FUNCTION_BLOCK FB_INFLUX_DB_ADS IMPLEMENTS I_INFLUXDB_ADS
VAR_IN_OUT
  bResult:                                                BOOL;
END_VAR
VAR_INPUT
  bADSLifeBit:                                            BOOL;
  bAdsConnected:                                          BOOL;
  bReady:                                                 BOOL;
  bBusy:                                                  BOOL;
END_VAR
VAR //General
	{attribute 'instance-path'} 
  {attribute 'noinit'} 
	strInstancePath:									                      STRING;
	bInit: 												                          BOOL:=TRUE;
	strFullObjectPath: 								                      STRING;
	stEvent:											                          ST_EVENT;
	bAck:												                            BOOL;
	
END_VAR
VAR   // From FB_init	
	itfOpMode:											                        I_OP_MODE; 
  itfEventLogger:                                         I_EVENT_LOGGER;
END_VAR                                      				
VAR	// Step chain control                				
  eSeq, eLastSeq, eNextSeq:					                      E_SEQ_DATABASE; 
  i:														                          INT;
  stSeqCtrlGeneral:											                  ST_SEQ_CTRL_GEN;     	
END_VAR                                             		
VAR                                                 		
	bMethodeFromExtStarted:									                BOOL;
	bMethodeFromExtActive:									                BOOL;
	bMethodeFromExtDone:									                  BOOL;
	strTemp:												                        STRING;
END_VAR   
VAR
  // From ADS
  bDBLifeBit:                                             BOOL;
  liDatabaseSizeInMb:                                     LINT;
  udiDatabaseSizeInMb:                                    UDINT;
  uiTotalMeasurements:                                    UINT;
  // To ADS
  bGetBucketExist:                                        BOOL;
  sBucketName:                                            T_MaxString := '3925-HZP';
  bGetMeasurementExist:                                   BOOL;
  sMeasurementName:                                       T_MaxString;
  bDeleteMeasurement:                                     BOOL;
  bDeleteAllMeasurements:                                 BOOL;
  bWriteStructData:                                       BOOL;
  sTagName:                                               T_MaxString;
  sFieldName:                                             T_MaxString;
  stFieldValues:                                          ST_DATABASE_RECORD;
  pFieldStructContent:                                    POINTER TO ARRAY [0..99] OF T_MaxString;
  pFieldNames:                                            POINTER TO ARRAY [0..99] OF T_MaxString;
  dtFrom:                                                 DT;
  dtTo:                                                   DT;
  sDtFrom:                                                T_MaxString;
  sDtTo:                                                  T_MaxString;
  sFieldNameExistCheck:                                   T_MaxString;
  bGetTagExist:                                           BOOL;
  bGetFieldExist:                                         BOOL;
  bClearMeasurement:                                      BOOL;
  bDeleteTag:                                             BOOL;
  bDeleteTagContentBlock:                                 BOOL;
  bDeleteField:                                           BOOL;
  bGetTotalMeasurements:                                  BOOL;
END_VAR    
VAR // State
  tLifeBitTimeout:                                        TIME := T#5S;
  // ADS
  uiADSStateSeq:                                          UINT := 0;
  tonADSState:                                            TON;
  bResetADSStateTimer:                                    BOOL;
  bADSState:                                              BOOL := TRUE;
  // InfluxDB
  uiInfluxDBStateSeq:                                     UINT := 0;
  tonInfluxDBState:                                       TON;
  bResetInfluxDBStateTimer:                               BOOL;
  bInfluxDBState:                                         BOOL := TRUE;
END_VAR              	
VAR_TEMP                    	
	iTemp:										                              INT;
END_VAR

// Set FBs and Interfaces ready after switch internal step
IF stSeqCtrlGeneral.iInternalSeqStateCase <> stSeqCtrlGeneral.iLastInternalSeqStateCase AND NOT stSeqCtrlGeneral.bExitSetReadyState THEN
  IF TRUE
  THEN
    stSeqCtrlGeneral.bExitSetReadyState := TRUE;
  ELSE
    RETURN;
  END_IF
END_IF

stSeqCtrlGeneral.strObject := F_CreateObjectName(strInstancePath);

// Init
// Format Time string for InfluxDB
sDtFrom := DT_TO_STRING(dtFrom);
sDtFrom := DELETE(sDtFrom, 3, 1);
sDtFrom := REPLACE(sDtFrom, 'T', 1, 11);
sDtFrom := CONCAT(sDtFrom, 'Z');
sDtTo := DT_TO_STRING(dtTo);
sDtTo := DELETE(sDtTo, 3, 1);
sDtTo := REPLACE(sDtTo, 'T', 1, 11);
sDtTo := CONCAT(sDtTo, 'Z');

// Actions
A_010_ADSState();
A_020_InfluxDBState();

// First method call
_m_SequenceManager();
//_m_SaveLastStep();

udiDatabaseSizeInMb := TO_UDINT(liDatabaseSizeInMb);

CASE eSeq OF 
  E_SEQ_DATABASE.BASE:;
  
	E_SEQ_DATABASE.INIT: _m_Seq_INIT();
		IF TRUE
		AND (stSeqCtrlGeneral.eActiveSeqState = E_SEQ_GENERAL.DONE) 
		THEN
			eSeq := E_SEQ_DATABASE.BASE;
		END_IF
		
	E_SEQ_DATABASE.SETUP:;
  
	// Process
  E_SEQ_DATABASE.BUCKET_EXIST_CHECK: _m_Seq_BUCKET_EXIST_CHECK();
    IF TRUE
		AND (stSeqCtrlGeneral.eActiveSeqState = E_SEQ_GENERAL.DONE) 
		THEN
			eSeq := E_SEQ_DATABASE.BASE;
		END_IF
  
	E_SEQ_DATABASE.MEASUREMENT_EXIST_CHECK:         _m_Seq_MEASUREMENT_EXIST_CHECK();
    IF TRUE
		AND (stSeqCtrlGeneral.eActiveSeqState = E_SEQ_GENERAL.DONE) 
		THEN
			eSeq := E_SEQ_DATABASE.BASE;
		END_IF
    
  E_SEQ_DATABASE.WRITE_STRUCT:  _m_Seq_WRITE_STRUCT();
    IF TRUE
		AND (stSeqCtrlGeneral.eActiveSeqState = E_SEQ_GENERAL.DONE) 
		THEN
			eSeq := E_SEQ_DATABASE.BASE;
		END_IF
  
  E_SEQ_DATABASE.TAG_EXIST_CHECK:     _m_Seq_TAG_EXIST_CHECK();
    IF TRUE
		AND (stSeqCtrlGeneral.eActiveSeqState = E_SEQ_GENERAL.DONE) 
		THEN
			eSeq := E_SEQ_DATABASE.BASE;
		END_IF
    
  E_SEQ_DATABASE.FIELD_EXIST_CHECK:     _m_Seq_FIELD_EXIST_CHECK();
    IF TRUE
		AND (stSeqCtrlGeneral.eActiveSeqState = E_SEQ_GENERAL.DONE) 
		THEN
			eSeq := E_SEQ_DATABASE.BASE;
		END_IF
    
  E_SEQ_DATABASE.DELETE_MEASUREMENT:    _m_Seq_DELETE_MEASUREMENT();
    IF TRUE
		AND (stSeqCtrlGeneral.eActiveSeqState = E_SEQ_GENERAL.DONE) 
		THEN
			eSeq := E_SEQ_DATABASE.BASE;
		END_IF
    
  E_SEQ_DATABASE.DELETE_ALL_MEASUREMENTS:    _m_Seq_DELETE_ALL_MEASUREMENTS();
    IF TRUE
		AND (stSeqCtrlGeneral.eActiveSeqState = E_SEQ_GENERAL.DONE) 
		THEN
			eSeq := E_SEQ_DATABASE.BASE;
		END_IF
  
  E_SEQ_DATABASE.DELETE_TAG:    _m_Seq_DELETE_TAG();
    IF TRUE
		AND (stSeqCtrlGeneral.eActiveSeqState = E_SEQ_GENERAL.DONE) 
		THEN
			eSeq := E_SEQ_DATABASE.BASE;
		END_IF
    
  E_SEQ_DATABASE.DELETE_TAG_CONTENT_BLOCK:    _m_Seq_DELETE_TAG_CONTENT_BLOCK();
    IF TRUE
		AND (stSeqCtrlGeneral.eActiveSeqState = E_SEQ_GENERAL.DONE) 
		THEN
			eSeq := E_SEQ_DATABASE.BASE;
		END_IF
  
  E_SEQ_DATABASE.DELETE_FIELD:           _m_Seq_DELETE_FIELD();
    IF TRUE
		AND (stSeqCtrlGeneral.eActiveSeqState = E_SEQ_GENERAL.DONE) 
		THEN
			eSeq := E_SEQ_DATABASE.BASE;
		END_IF
    
  E_SEQ_DATABASE.GET_TOTAL_MEASUREMENTS:           _m_Seq_GET_TOTAL_MEASUREMENTS();
    IF TRUE
		AND (stSeqCtrlGeneral.eActiveSeqState = E_SEQ_GENERAL.DONE) 
		THEN
			eSeq := E_SEQ_DATABASE.BASE;
		END_IF

  // End
	E_SEQ_DATABASE.END:;
	E_SEQ_DATABASE.ERROR_SEQ:;	
END_CASE

strTemp:=TO_STRING(eSeq);

METHOD PRIVATE _m_DebugManager
VAR_INPUT
	iStepID: int;
END_VAR
IF TRUE
AND THIS^.stSeqCtrlGeneral.bDebugModeActive 
AND NOT THIS^.stSeqCtrlGeneral.bActiveStep
THEN


THIS^.stSeqCtrlGeneral.bBreakpointActive:=FALSE;

FOR i:=0 TO 10 DO
	
	IF TRUE
	AND iStepID=THIS^.stSeqCtrlGeneral.listBreakpoint[i] 
	AND iStepID<>0
	THEN
		EXIT;
	END_IF
END_FOR
IF (i<=10) THEN
	THIS^.stSeqCtrlGeneral.bBreakpointActive:=TRUE;
END_IF

END_IF
END_METHOD

METHOD PRIVATE _m_Delay : BOOL
VAR_INPUT
	DelayTime:	TIME;
END_VAR
THIS^.stSeqCtrlGeneral.bDelayActive:=TRUE;
THIS^.stSeqCtrlGeneral.tDelay:=DelayTime;
_m_Delay:=FALSE;
IF THIS^.stSeqCtrlGeneral.tonDelay.Q THEN
	_m_Delay:=TRUE;
END_IF
END_METHOD

METHOD PRIVATE _m_GeneralStepSetting : BOOL
VAR_INPUT
	StepType:			    	E_STEP_STATE_TYPE;
	InfoTextID:					STRING(20);
	EnableDebug:	   			BOOL;	
	
END_VAR
IF THIS^.stSeqCtrlGeneral.bActiveStep THEN
	THIS^.stSeqCtrlGeneral.eStep_Type:=StepType;
	THIS^.stSeqCtrlGeneral.strExtraInfo:= GenLib.F_RET_TXTLIST_ENTRY(strPortNr:='851',strID:='',strTxtLstName:=InfoTextID);
END_IF
END_METHOD

METHOD PRIVATE _m_SaveLastStep : BOOL
VAR_INPUT
END_VAR
VAR
	i: dint;
END_VAR
IF NOT THIS^.stSeqCtrlGeneral.bActiveStep THEN
	
	FOR i:=49 TO 1 BY -1 DO
			stSeqCtrlGeneral.listLastSteps[i].strStepName:=stSeqCtrlGeneral.listLastSteps[i-1].strStepName;
			stSeqCtrlGeneral.listLastSteps[i].tStepTime:=stSeqCtrlGeneral.listLastSteps[i-1].tStepTime;
			stSeqCtrlGeneral.listLastSteps[i].tDelayTime:=stSeqCtrlGeneral.listLastSteps[i-1].tDelayTime;
	END_FOR
	stSeqCtrlGeneral.listLastSteps[0].strStepName:=TO_STRING(THIS^.eSeq);
	stSeqCtrlGeneral.listLastSteps[1].tStepTime:=THIS^.stSeqCtrlGeneral.tonStepTime.ET;
	stSeqCtrlGeneral.listLastSteps[1].tStepTime:=THIS^.stSeqCtrlGeneral.tonDelay.ET;
ELSE
	stSeqCtrlGeneral.listLastSteps[0].tStepTime:=THIS^.stSeqCtrlGeneral.tonStepTime.ET;
	stSeqCtrlGeneral.listLastSteps[0].tDelayTime:=THIS^.stSeqCtrlGeneral.tonDelay.ET;	
END_IF
END_METHOD

METHOD PRIVATE _m_Seq_BUCKET_EXIST_CHECK : E_SEQ_PROCESS
VAR_INPUT
END_VAR
VAR
	ActiveSeq: STRING;
END_VAR
//THIS^._m_GeneralStepSetting(StepType:=E_STEP_STATE_TYPE.INIT,
ActiveSeq := TO_STRING(THIS^.eSeq);

CASE THIS^.stSeqCtrlGeneral.eActiveSeqState OF
E_SEQ_GENERAL.READY:;
	
E_SEQ_GENERAL.EXECUTE:;
	IF TRUE
	THEN
		THIS^.stSeqCtrlGeneral.eActiveSeqState := E_SEQ_GENERAL.RESET;
	END_IF
  
E_SEQ_GENERAL.RESET:;
	THIS^.stSeqCtrlGeneral.iInternalSeqStateCase := 0;
	IF TRUE
	THEN
    THIS^.bResult := FALSE;
		THIS^.stSeqCtrlGeneral.eActiveSeqState := E_SEQ_GENERAL.BUSY;
	END_IF
  
E_SEQ_GENERAL.BUSY:;
	CASE THIS^.stSeqCtrlGeneral.iInternalSeqStateCase OF
    0:  // Execute
      IF TRUE 
      AND THIS^.bAdsConnected
      AND NOT THIS^.bBusy
      AND THIS^.bReady
			THEN 
        THIS^.bGetBucketExist := TRUE;
        THIS^.stSeqCtrlGeneral.iInternalSeqStateCase := 10;
			END_IF

    10:	// Wait for done
      IF TRUE 
      AND NOT THIS^.bBusy
      AND THIS^.bReady
      AND NOT THIS^.bGetBucketExist
			THEN 
        THIS^.stSeqCtrlGeneral.iInternalSeqStateCase := 1000;
			END_IF
      
    1000: // Exit step
      IF TRUE
      THEN
        THIS^.stSeqCtrlGeneral.iInternalSeqStateCase := 9999;
			END_IF
      
	ELSE
		THIS^.stSeqCtrlGeneral.eActiveSeqState := E_SEQ_GENERAL.DONE;  
	END_CASE
	THIS^.stSeqCtrlGeneral.strExtraInfo := CONCAT('Internal state: ', TO_STRING(THIS^.stSeqCtrlGeneral.iInternalSeqStateCase));

E_SEQ_GENERAL.DONE:;

E_SEQ_GENERAL.ERROR:;

E_SEQ_GENERAL.TIME_OUT:; 

ELSE
  THIS^.stSeqCtrlGeneral.eActiveSeqState := E_SEQ_GENERAL.ERROR;
END_CASE
END_METHOD

METHOD PRIVATE _m_Seq_CLEAR_MEASUREMENT : E_SEQ_PROCESS
VAR_INPUT
END_VAR
VAR
	ActiveSeq: STRING;
END_VAR
//THIS^._m_GeneralStepSetting(StepType:=E_STEP_STATE_TYPE.INIT,
ActiveSeq := TO_STRING(THIS^.eSeq);

CASE THIS^.stSeqCtrlGeneral.eActiveSeqState OF
E_SEQ_GENERAL.READY:;
	
E_SEQ_GENERAL.EXECUTE:;
	IF TRUE
	THEN
		THIS^.stSeqCtrlGeneral.eActiveSeqState := E_SEQ_GENERAL.RESET;
	END_IF
  
E_SEQ_GENERAL.RESET:;
	THIS^.stSeqCtrlGeneral.iInternalSeqStateCase := 0;
	IF TRUE
	THEN
    THIS^.bResult := FALSE;
		THIS^.stSeqCtrlGeneral.eActiveSeqState := E_SEQ_GENERAL.BUSY;
	END_IF
  
E_SEQ_GENERAL.BUSY:;
	CASE THIS^.stSeqCtrlGeneral.iInternalSeqStateCase OF
		0:	// Entrance step --> Create command
      IF TRUE 
      AND THIS^.bAdsConnected
      AND NOT THIS^.bBusy
      AND THIS^.bReady
			THEN 
        THIS^.bClearMeasurement := TRUE;
        THIS^.stSeqCtrlGeneral.iInternalSeqStateCase := 10;
			END_IF
      
    10:	// Wait for done
      IF TRUE 
      AND NOT THIS^.bBusy
      AND THIS^.bReady
      AND NOT THIS^.bClearMeasurement
			THEN 
        THIS^.stSeqCtrlGeneral.iInternalSeqStateCase := 1000;
			END_IF
      
    1000: // Exit step
      IF TRUE
      THEN
        THIS^.stSeqCtrlGeneral.iInternalSeqStateCase := 9999;
			END_IF
      
	ELSE
		THIS^.stSeqCtrlGeneral.eActiveSeqState := E_SEQ_GENERAL.DONE;  
	END_CASE
	THIS^.stSeqCtrlGeneral.strExtraInfo := CONCAT('Internal state: ', TO_STRING(THIS^.stSeqCtrlGeneral.iInternalSeqStateCase));

E_SEQ_GENERAL.DONE:;

E_SEQ_GENERAL.ERROR:;

E_SEQ_GENERAL.TIME_OUT:; 
IF TRUE
AND THIS^.stSeqCtrlGeneral.bTimeOutActiveQuit 
THEN
  THIS^.stSeqCtrlGeneral.strExtraInfo := 'Bitte quittieren und erneut testen';
  IF TRUE
  //AND itfOpMode.P_QUIT
  THEN
    THIS^.stSeqCtrlGeneral.eActiveSeqState := E_SEQ_GENERAL.EXECUTE;
	END_IF
  
END_IF

ELSE
  THIS^.stSeqCtrlGeneral.eActiveSeqState := E_SEQ_GENERAL.ERROR;
END_CASE
END_METHOD

METHOD PRIVATE _m_Seq_DELETE_ALL_MEASUREMENTS : E_SEQ_PROCESS
VAR_INPUT
END_VAR
VAR
	ActiveSeq: STRING;
END_VAR
//THIS^._m_GeneralStepSetting(StepType:=E_STEP_STATE_TYPE.INIT,
ActiveSeq := TO_STRING(THIS^.eSeq);

CASE THIS^.stSeqCtrlGeneral.eActiveSeqState OF
E_SEQ_GENERAL.READY:;

E_SEQ_GENERAL.EXECUTE:;
	IF TRUE
	THEN
		THIS^.stSeqCtrlGeneral.eActiveSeqState := E_SEQ_GENERAL.RESET;
	END_IF
  
E_SEQ_GENERAL.RESET:;
	THIS^.stSeqCtrlGeneral.iInternalSeqStateCase := 0;
	IF TRUE
	THEN
    THIS^.bResult := FALSE;
		THIS^.stSeqCtrlGeneral.eActiveSeqState := E_SEQ_GENERAL.BUSY;
	END_IF
  
E_SEQ_GENERAL.BUSY:;
	CASE THIS^.stSeqCtrlGeneral.iInternalSeqStateCase OF
		0:	// Entrance step --> Create command
      IF TRUE 
      AND THIS^.bAdsConnected
      AND NOT THIS^.bBusy
      AND THIS^.bReady
			THEN 
        THIS^.bDeleteAllMeasurements := TRUE;
        THIS^.stSeqCtrlGeneral.iInternalSeqStateCase := 10;
			END_IF
      
    10:	// Wait for done
      IF TRUE 
      AND NOT THIS^.bBusy
      AND THIS^.bReady
      AND NOT THIS^.bDeleteAllMeasurements
			THEN 
        THIS^.stSeqCtrlGeneral.iInternalSeqStateCase := 1000;
			END_IF
      
    1000: // Exit step
      IF TRUE
      THEN
        THIS^.stSeqCtrlGeneral.iInternalSeqStateCase := 9999;
			END_IF
      
	ELSE
		THIS^.stSeqCtrlGeneral.eActiveSeqState := E_SEQ_GENERAL.DONE;  
	END_CASE
	THIS^.stSeqCtrlGeneral.strExtraInfo := CONCAT('Internal state: ', TO_STRING(THIS^.stSeqCtrlGeneral.iInternalSeqStateCase));

E_SEQ_GENERAL.DONE:;

E_SEQ_GENERAL.ERROR:;

E_SEQ_GENERAL.TIME_OUT:; 
IF TRUE
AND THIS^.stSeqCtrlGeneral.bTimeOutActiveQuit 
THEN
  THIS^.stSeqCtrlGeneral.strExtraInfo := 'Bitte quittieren und erneut testen';
  IF TRUE
  //AND itfOpMode.P_QUIT
  THEN
    THIS^.stSeqCtrlGeneral.eActiveSeqState := E_SEQ_GENERAL.EXECUTE;
	END_IF
  
END_IF

ELSE
  THIS^.stSeqCtrlGeneral.eActiveSeqState := E_SEQ_GENERAL.ERROR;
END_CASE
END_METHOD

METHOD PRIVATE _m_Seq_DELETE_FIELD : E_SEQ_PROCESS
VAR_INPUT
END_VAR
VAR
	ActiveSeq: STRING;
END_VAR
//THIS^._m_GeneralStepSetting(StepType:=E_STEP_STATE_TYPE.INIT,
ActiveSeq := TO_STRING(THIS^.eSeq);

CASE THIS^.stSeqCtrlGeneral.eActiveSeqState OF
E_SEQ_GENERAL.READY:;
	
E_SEQ_GENERAL.EXECUTE:;
	IF TRUE
	THEN
		THIS^.stSeqCtrlGeneral.eActiveSeqState := E_SEQ_GENERAL.RESET;
	END_IF
  
E_SEQ_GENERAL.RESET:;
	THIS^.stSeqCtrlGeneral.iInternalSeqStateCase := 0;
	IF TRUE
	THEN
    THIS^.bResult := FALSE;
		THIS^.stSeqCtrlGeneral.eActiveSeqState := E_SEQ_GENERAL.BUSY;
	END_IF
  
E_SEQ_GENERAL.BUSY:;
	CASE THIS^.stSeqCtrlGeneral.iInternalSeqStateCase OF
    0:  // Execute
      IF TRUE 
      AND THIS^.bAdsConnected
      AND NOT THIS^.bBusy
      AND THIS^.bReady
			THEN 
        THIS^.bDeleteField := TRUE;
        THIS^.stSeqCtrlGeneral.iInternalSeqStateCase := 10;
			END_IF

    10:	// Wait for done
      IF TRUE 
      AND NOT THIS^.bBusy
      AND THIS^.bReady
      AND NOT THIS^.bDeleteField
			THEN 
        THIS^.stSeqCtrlGeneral.iInternalSeqStateCase := 1000;
			END_IF
      
    1000: // Exit step
      IF TRUE
      THEN
        THIS^.stSeqCtrlGeneral.iInternalSeqStateCase := 9999;
			END_IF
      
	ELSE
		THIS^.stSeqCtrlGeneral.eActiveSeqState := E_SEQ_GENERAL.DONE;  
	END_CASE
	THIS^.stSeqCtrlGeneral.strExtraInfo := CONCAT('Internal state: ', TO_STRING(THIS^.stSeqCtrlGeneral.iInternalSeqStateCase));

E_SEQ_GENERAL.DONE:;

E_SEQ_GENERAL.ERROR:;

E_SEQ_GENERAL.TIME_OUT:; 

ELSE
  THIS^.stSeqCtrlGeneral.eActiveSeqState := E_SEQ_GENERAL.ERROR;
END_CASE
END_METHOD

METHOD PRIVATE _m_Seq_DELETE_MEASUREMENT : E_SEQ_PROCESS
VAR_INPUT
END_VAR
VAR
	ActiveSeq: STRING;
END_VAR
//THIS^._m_GeneralStepSetting(StepType:=E_STEP_STATE_TYPE.INIT,
ActiveSeq := TO_STRING(THIS^.eSeq);

CASE THIS^.stSeqCtrlGeneral.eActiveSeqState OF
E_SEQ_GENERAL.READY:;
	
E_SEQ_GENERAL.EXECUTE:;
	IF TRUE
	THEN
		THIS^.stSeqCtrlGeneral.eActiveSeqState := E_SEQ_GENERAL.RESET;
	END_IF
  
E_SEQ_GENERAL.RESET:;
	THIS^.stSeqCtrlGeneral.iInternalSeqStateCase := 0;
	IF TRUE
	THEN
    THIS^.bResult := FALSE;
		THIS^.stSeqCtrlGeneral.eActiveSeqState := E_SEQ_GENERAL.BUSY;
	END_IF
  
E_SEQ_GENERAL.BUSY:;
	CASE THIS^.stSeqCtrlGeneral.iInternalSeqStateCase OF
		0:	// Entrance step --> Create command
      IF TRUE 
      AND THIS^.bAdsConnected
      AND NOT THIS^.bBusy
      AND THIS^.bReady
			THEN 
        THIS^.bDeleteMeasurement := TRUE;
        THIS^.stSeqCtrlGeneral.iInternalSeqStateCase := 10;
			END_IF
      
    10:	// Wait for done
      IF TRUE 
      AND NOT THIS^.bBusy
      AND THIS^.bReady
      AND NOT THIS^.bDeleteMeasurement
			THEN 
        THIS^.stSeqCtrlGeneral.iInternalSeqStateCase := 1000;
			END_IF
      
    1000: // Exit step
      IF TRUE
      THEN
        THIS^.stSeqCtrlGeneral.iInternalSeqStateCase := 9999;
			END_IF
      
	ELSE
		THIS^.stSeqCtrlGeneral.eActiveSeqState := E_SEQ_GENERAL.DONE;  
	END_CASE
	THIS^.stSeqCtrlGeneral.strExtraInfo := CONCAT('Internal state: ', TO_STRING(THIS^.stSeqCtrlGeneral.iInternalSeqStateCase));

E_SEQ_GENERAL.DONE:;

E_SEQ_GENERAL.ERROR:;

E_SEQ_GENERAL.TIME_OUT:; 
IF TRUE
AND THIS^.stSeqCtrlGeneral.bTimeOutActiveQuit 
THEN
  THIS^.stSeqCtrlGeneral.strExtraInfo := 'Bitte quittieren und erneut testen';
  IF TRUE
  //AND itfOpMode.P_QUIT
  THEN
    THIS^.stSeqCtrlGeneral.eActiveSeqState := E_SEQ_GENERAL.EXECUTE;
	END_IF
  
END_IF

ELSE
  THIS^.stSeqCtrlGeneral.eActiveSeqState := E_SEQ_GENERAL.ERROR;
END_CASE
END_METHOD

METHOD PRIVATE _m_Seq_DELETE_TAG : E_SEQ_PROCESS
VAR_INPUT
END_VAR
VAR
	ActiveSeq: STRING;
END_VAR
//THIS^._m_GeneralStepSetting(StepType:=E_STEP_STATE_TYPE.INIT,
ActiveSeq := TO_STRING(THIS^.eSeq);

CASE THIS^.stSeqCtrlGeneral.eActiveSeqState OF
E_SEQ_GENERAL.READY:;
	
E_SEQ_GENERAL.EXECUTE:;
	IF TRUE
	THEN
		THIS^.stSeqCtrlGeneral.eActiveSeqState := E_SEQ_GENERAL.RESET;
	END_IF
  
E_SEQ_GENERAL.RESET:;
	THIS^.stSeqCtrlGeneral.iInternalSeqStateCase := 0;
	IF TRUE
	THEN
    THIS^.bResult := FALSE;
		THIS^.stSeqCtrlGeneral.eActiveSeqState := E_SEQ_GENERAL.BUSY;
	END_IF
  
E_SEQ_GENERAL.BUSY:;
	CASE THIS^.stSeqCtrlGeneral.iInternalSeqStateCase OF
    0:  // Execute
      IF TRUE 
      AND THIS^.bAdsConnected
      AND NOT THIS^.bBusy
      AND THIS^.bReady
			THEN 
        THIS^.bDeleteTag := TRUE;
        THIS^.stSeqCtrlGeneral.iInternalSeqStateCase := 10;
			END_IF

    10:	// Wait for done
      IF TRUE 
      AND NOT THIS^.bBusy
      AND THIS^.bReady
      AND NOT THIS^.bDeleteTag
			THEN 
        THIS^.stSeqCtrlGeneral.iInternalSeqStateCase := 1000;
			END_IF
      
    1000: // Exit step
      IF TRUE
      THEN
        THIS^.stSeqCtrlGeneral.iInternalSeqStateCase := 9999;
			END_IF
      
	ELSE
		THIS^.stSeqCtrlGeneral.eActiveSeqState := E_SEQ_GENERAL.DONE;  
	END_CASE
	THIS^.stSeqCtrlGeneral.strExtraInfo := CONCAT('Internal state: ', TO_STRING(THIS^.stSeqCtrlGeneral.iInternalSeqStateCase));

E_SEQ_GENERAL.DONE:;

E_SEQ_GENERAL.ERROR:;

E_SEQ_GENERAL.TIME_OUT:; 

ELSE
  THIS^.stSeqCtrlGeneral.eActiveSeqState := E_SEQ_GENERAL.ERROR;
END_CASE
END_METHOD

METHOD PRIVATE _m_Seq_DELETE_TAG_CONTENT_BLOCK : E_SEQ_PROCESS
VAR_INPUT
END_VAR
VAR
	ActiveSeq: STRING;
END_VAR
//THIS^._m_GeneralStepSetting(StepType:=E_STEP_STATE_TYPE.INIT,
ActiveSeq := TO_STRING(THIS^.eSeq);

CASE THIS^.stSeqCtrlGeneral.eActiveSeqState OF
E_SEQ_GENERAL.READY:;
	
E_SEQ_GENERAL.EXECUTE:;
	IF TRUE
	THEN
		THIS^.stSeqCtrlGeneral.eActiveSeqState := E_SEQ_GENERAL.RESET;
	END_IF
  
E_SEQ_GENERAL.RESET:;
	THIS^.stSeqCtrlGeneral.iInternalSeqStateCase := 0;
	IF TRUE
	THEN
    THIS^.bResult := FALSE;
		THIS^.stSeqCtrlGeneral.eActiveSeqState := E_SEQ_GENERAL.BUSY;
	END_IF
  
E_SEQ_GENERAL.BUSY:;
	CASE THIS^.stSeqCtrlGeneral.iInternalSeqStateCase OF
    0:  // Execute
      IF TRUE 
      AND THIS^.bAdsConnected
      AND NOT THIS^.bBusy
      AND THIS^.bReady
			THEN 
        THIS^.bDeleteTagContentBlock := TRUE;
        THIS^.stSeqCtrlGeneral.iInternalSeqStateCase := 10;
			END_IF

    10:	// Wait for done
      IF TRUE 
      AND NOT THIS^.bBusy
      AND THIS^.bReady
      AND NOT THIS^.bDeleteTagContentBlock
			THEN 
        THIS^.stSeqCtrlGeneral.iInternalSeqStateCase := 1000;
			END_IF
      
    1000: // Exit step
      IF TRUE
      THEN
        THIS^.stSeqCtrlGeneral.iInternalSeqStateCase := 9999;
			END_IF
      
	ELSE
		THIS^.stSeqCtrlGeneral.eActiveSeqState := E_SEQ_GENERAL.DONE;  
	END_CASE
	THIS^.stSeqCtrlGeneral.strExtraInfo := CONCAT('Internal state: ', TO_STRING(THIS^.stSeqCtrlGeneral.iInternalSeqStateCase));

E_SEQ_GENERAL.DONE:;

E_SEQ_GENERAL.ERROR:;

E_SEQ_GENERAL.TIME_OUT:; 

ELSE
  THIS^.stSeqCtrlGeneral.eActiveSeqState := E_SEQ_GENERAL.ERROR;
END_CASE
END_METHOD

METHOD PRIVATE _m_Seq_FIELD_EXIST_CHECK : E_SEQ_PROCESS
VAR_INPUT
END_VAR
VAR
	ActiveSeq: STRING;
END_VAR
//THIS^._m_GeneralStepSetting(StepType:=E_STEP_STATE_TYPE.INIT,
ActiveSeq := TO_STRING(THIS^.eSeq);

CASE THIS^.stSeqCtrlGeneral.eActiveSeqState OF
E_SEQ_GENERAL.READY:;
	
E_SEQ_GENERAL.EXECUTE:;
	IF TRUE
	THEN
		THIS^.stSeqCtrlGeneral.eActiveSeqState := E_SEQ_GENERAL.RESET;
	END_IF
  
E_SEQ_GENERAL.RESET:;
	THIS^.stSeqCtrlGeneral.iInternalSeqStateCase := 0;
	IF TRUE
	THEN
    THIS^.bResult := FALSE;
		THIS^.stSeqCtrlGeneral.eActiveSeqState := E_SEQ_GENERAL.BUSY;
	END_IF
  
E_SEQ_GENERAL.BUSY:;
	CASE THIS^.stSeqCtrlGeneral.iInternalSeqStateCase OF
    0:  // Execute
      IF TRUE 
      AND THIS^.bAdsConnected
      AND NOT THIS^.bBusy
      AND THIS^.bReady
			THEN 
        THIS^.bGetFieldExist := TRUE;
        THIS^.stSeqCtrlGeneral.iInternalSeqStateCase := 10;
			END_IF

    10:	// Wait for done
      IF TRUE 
      AND NOT THIS^.bBusy
      AND THIS^.bReady
      AND NOT THIS^.bGetFieldExist
			THEN 
        THIS^.stSeqCtrlGeneral.iInternalSeqStateCase := 1000;
			END_IF
      
    1000: // Exit step
      IF TRUE
      THEN
        THIS^.stSeqCtrlGeneral.iInternalSeqStateCase := 9999;
			END_IF
      
	ELSE
		THIS^.stSeqCtrlGeneral.eActiveSeqState := E_SEQ_GENERAL.DONE;  
	END_CASE
	THIS^.stSeqCtrlGeneral.strExtraInfo := CONCAT('Internal state: ', TO_STRING(THIS^.stSeqCtrlGeneral.iInternalSeqStateCase));

E_SEQ_GENERAL.DONE:;

E_SEQ_GENERAL.ERROR:;

E_SEQ_GENERAL.TIME_OUT:; 

ELSE
  THIS^.stSeqCtrlGeneral.eActiveSeqState := E_SEQ_GENERAL.ERROR;
END_CASE
END_METHOD

METHOD PRIVATE _m_Seq_GET_TOTAL_MEASUREMENTS : E_SEQ_PROCESS
VAR_INPUT
END_VAR
VAR
	ActiveSeq: STRING;
END_VAR
//THIS^._m_GeneralStepSetting(StepType:=E_STEP_STATE_TYPE.INIT,
ActiveSeq := TO_STRING(THIS^.eSeq);

CASE THIS^.stSeqCtrlGeneral.eActiveSeqState OF
E_SEQ_GENERAL.READY:;
	
E_SEQ_GENERAL.EXECUTE:;
	IF TRUE
	THEN
		THIS^.stSeqCtrlGeneral.eActiveSeqState := E_SEQ_GENERAL.RESET;
	END_IF
  
E_SEQ_GENERAL.RESET:;
	THIS^.stSeqCtrlGeneral.iInternalSeqStateCase := 0;
	IF TRUE
	THEN
    THIS^.bResult := FALSE;
		THIS^.stSeqCtrlGeneral.eActiveSeqState := E_SEQ_GENERAL.BUSY;
	END_IF
  
E_SEQ_GENERAL.BUSY:;
	CASE THIS^.stSeqCtrlGeneral.iInternalSeqStateCase OF
    0:  // Execute
      IF TRUE 
      AND THIS^.bAdsConnected
      AND NOT THIS^.bBusy
      AND THIS^.bReady
			THEN 
        THIS^.bGetTotalMeasurements := TRUE;
        THIS^.stSeqCtrlGeneral.iInternalSeqStateCase := 10;
			END_IF

    10:	// Wait for done
      IF TRUE 
      AND NOT THIS^.bBusy
      AND THIS^.bReady
      AND NOT THIS^.bGetTotalMeasurements
			THEN 
        THIS^.stSeqCtrlGeneral.iInternalSeqStateCase := 1000;
			END_IF
      
    1000: // Exit step
      IF TRUE
      THEN
        THIS^.stSeqCtrlGeneral.iInternalSeqStateCase := 9999;
			END_IF
      
	ELSE
		THIS^.stSeqCtrlGeneral.eActiveSeqState := E_SEQ_GENERAL.DONE;  
	END_CASE
	THIS^.stSeqCtrlGeneral.strExtraInfo := CONCAT('Internal state: ', TO_STRING(THIS^.stSeqCtrlGeneral.iInternalSeqStateCase));

E_SEQ_GENERAL.DONE:;

E_SEQ_GENERAL.ERROR:;

E_SEQ_GENERAL.TIME_OUT:; 

ELSE
  THIS^.stSeqCtrlGeneral.eActiveSeqState := E_SEQ_GENERAL.ERROR;
END_CASE
END_METHOD

METHOD PRIVATE _m_Seq_INIT : E_SEQ_PROCESS
VAR_INPUT
END_VAR
VAR
	ActiveSeq: STRING;
END_VAR
VAR
	
END_VAR
//THIS^._m_GeneralStepSetting(StepType:=E_STEP_STATE_TYPE.INIT,
ActiveSeq := TO_STRING(THIS^.eSeq);

CASE THIS^.stSeqCtrlGeneral.eActiveSeqState OF
E_SEQ_GENERAL.READY:;
	
E_SEQ_GENERAL.EXECUTE:;
	IF TRUE
	THEN
		THIS^.stSeqCtrlGeneral.eActiveSeqState := E_SEQ_GENERAL.RESET;
	END_IF
E_SEQ_GENERAL.RESET:;
	THIS^.stSeqCtrlGeneral.iInternalSeqStateCase := 0;
	IF TRUE
	THEN
		THIS^.stSeqCtrlGeneral.eActiveSeqState := E_SEQ_GENERAL.BUSY;
	END_IF
E_SEQ_GENERAL.BUSY:;
	CASE THIS^.stSeqCtrlGeneral.iInternalSeqStateCase OF
		0:	// Entrance step
      IF TRUE
			THEN 
        THIS^.bResult := FALSE;
        THIS^.bGetBucketExist := FALSE;
        THIS^.sBucketName := '';
        THIS^.bGetMeasurementExist := FALSE;
        THIS^.sMeasurementName := '';
        THIS^.bDeleteMeasurement := FALSE;
        THIS^.bDeleteAllMeasurements := FALSE;
        THIS^.bWriteStructData := FALSE;
        THIS^.sTagName := '';
        THIS^.sFieldName := '';
        //THIS^.stFieldValues := '';
        //FOR THIS^.i := 0 TO TO_INT(SIZEOF(arrFieldNames)) BY 1 DO
        //  THIS^.arrFieldNames[i] := '';
        //  THIS^.arrFieldStructContent[i] := '';
        //END_FOR
        THIS^.dtFrom := DT#1970-1-1-0:0:0;
        THIS^.dtTo := DT#1970-1-1-0:0:0;
				THIS^.stSeqCtrlGeneral.iInternalSeqStateCase := 1000;
			END_IF
      
    1000:	// Exit step
      IF TRUE
			THEN
        THIS^.stSeqCtrlGeneral.iInternalSeqStateCase := 9999;
      END_IF
      
	ELSE
		THIS^.stSeqCtrlGeneral.eActiveSeqState := E_SEQ_GENERAL.DONE;  
	END_CASE
	THIS^.stSeqCtrlGeneral.strExtraInfo := CONCAT('Internal state: ', TO_STRING(THIS^.stSeqCtrlGeneral.iInternalSeqStateCase));
E_SEQ_GENERAL.DONE:;
E_SEQ_GENERAL.ERROR:;
E_SEQ_GENERAL.TIME_OUT:; 

IF TRUE
AND THIS^.stSeqCtrlGeneral.bTimeOutActiveQuit 
THEN
  THIS^.stSeqCtrlGeneral.strExtraInfo := 'Bitte quittieren und erneut testen';
  IF TRUE
  //AND itfOpMode.P_QUIT
  THEN
    THIS^.stSeqCtrlGeneral.eActiveSeqState := E_SEQ_GENERAL.EXECUTE;
	END_IF
  
END_IF

ELSE
  THIS^.stSeqCtrlGeneral.eActiveSeqState := E_SEQ_GENERAL.ERROR;
END_CASE
END_METHOD

METHOD PRIVATE _m_Seq_MEASUREMENT_EXIST_CHECK : E_SEQ_PROCESS
VAR_INPUT
END_VAR
VAR
	ActiveSeq: STRING;
END_VAR
//THIS^._m_GeneralStepSetting(StepType:=E_STEP_STATE_TYPE.INIT,
ActiveSeq := TO_STRING(THIS^.eSeq);

CASE THIS^.stSeqCtrlGeneral.eActiveSeqState OF
E_SEQ_GENERAL.READY:;
	
E_SEQ_GENERAL.EXECUTE:;
	IF TRUE
	THEN
		THIS^.stSeqCtrlGeneral.eActiveSeqState := E_SEQ_GENERAL.RESET;
	END_IF
  
E_SEQ_GENERAL.RESET:;
	THIS^.stSeqCtrlGeneral.iInternalSeqStateCase := 0;
	IF TRUE
	THEN
    THIS^.bResult := FALSE;
		THIS^.stSeqCtrlGeneral.eActiveSeqState := E_SEQ_GENERAL.BUSY;
	END_IF
  
E_SEQ_GENERAL.BUSY:;
	CASE THIS^.stSeqCtrlGeneral.iInternalSeqStateCase OF
    0:  // Execute
      IF TRUE 
      AND THIS^.bAdsConnected
      AND NOT THIS^.bBusy
      AND THIS^.bReady
			THEN 
        THIS^.bGetMeasurementExist := TRUE;
        THIS^.stSeqCtrlGeneral.iInternalSeqStateCase := 10;
			END_IF

    10:	// Wait for done
      IF TRUE 
      AND NOT THIS^.bBusy
      AND THIS^.bReady
      AND NOT THIS^.bGetMeasurementExist
			THEN 
        THIS^.stSeqCtrlGeneral.iInternalSeqStateCase := 1000;
			END_IF
      
    1000: // Exit step
      IF TRUE
      THEN
        THIS^.stSeqCtrlGeneral.iInternalSeqStateCase := 9999;
			END_IF
      
	ELSE
		THIS^.stSeqCtrlGeneral.eActiveSeqState := E_SEQ_GENERAL.DONE;  
	END_CASE
	THIS^.stSeqCtrlGeneral.strExtraInfo := CONCAT('Internal state: ', TO_STRING(THIS^.stSeqCtrlGeneral.iInternalSeqStateCase));

E_SEQ_GENERAL.DONE:;

E_SEQ_GENERAL.ERROR:;

E_SEQ_GENERAL.TIME_OUT:; 

ELSE
  THIS^.stSeqCtrlGeneral.eActiveSeqState := E_SEQ_GENERAL.ERROR;
END_CASE
END_METHOD

METHOD PRIVATE _m_Seq_TAG_EXIST_CHECK : E_SEQ_PROCESS
VAR_INPUT
END_VAR
VAR
	ActiveSeq: STRING;
END_VAR
//THIS^._m_GeneralStepSetting(StepType:=E_STEP_STATE_TYPE.INIT,
ActiveSeq := TO_STRING(THIS^.eSeq);

CASE THIS^.stSeqCtrlGeneral.eActiveSeqState OF
E_SEQ_GENERAL.READY:;
	
E_SEQ_GENERAL.EXECUTE:;
	IF TRUE
	THEN
		THIS^.stSeqCtrlGeneral.eActiveSeqState := E_SEQ_GENERAL.RESET;
	END_IF
  
E_SEQ_GENERAL.RESET:;
	THIS^.stSeqCtrlGeneral.iInternalSeqStateCase := 0;
	IF TRUE
	THEN
    THIS^.bResult := FALSE;
		THIS^.stSeqCtrlGeneral.eActiveSeqState := E_SEQ_GENERAL.BUSY;
	END_IF
  
E_SEQ_GENERAL.BUSY:;
	CASE THIS^.stSeqCtrlGeneral.iInternalSeqStateCase OF
    0:  // Execute
      IF TRUE 
      AND THIS^.bAdsConnected
      AND NOT THIS^.bBusy
      AND THIS^.bReady
			THEN 
        THIS^.bGetTagExist := TRUE;
        THIS^.stSeqCtrlGeneral.iInternalSeqStateCase := 10;
			END_IF

    10:	// Wait for done
      IF TRUE 
      AND NOT THIS^.bBusy
      AND THIS^.bReady
      AND NOT THIS^.bGetTagExist
			THEN 
        THIS^.stSeqCtrlGeneral.iInternalSeqStateCase := 1000;
			END_IF
      
    1000: // Exit step
      IF TRUE
      THEN
        THIS^.stSeqCtrlGeneral.iInternalSeqStateCase := 9999;
			END_IF
      
	ELSE
		THIS^.stSeqCtrlGeneral.eActiveSeqState := E_SEQ_GENERAL.DONE;  
	END_CASE
	THIS^.stSeqCtrlGeneral.strExtraInfo := CONCAT('Internal state: ', TO_STRING(THIS^.stSeqCtrlGeneral.iInternalSeqStateCase));

E_SEQ_GENERAL.DONE:;

E_SEQ_GENERAL.ERROR:;

E_SEQ_GENERAL.TIME_OUT:; 

ELSE
  THIS^.stSeqCtrlGeneral.eActiveSeqState := E_SEQ_GENERAL.ERROR;
END_CASE
END_METHOD

METHOD PRIVATE _m_Seq_WRITE_STRUCT : E_SEQ_PROCESS
VAR_INPUT
END_VAR
VAR
	ActiveSeq: STRING;
END_VAR
//THIS^._m_GeneralStepSetting(StepType:=E_STEP_STATE_TYPE.INIT,
ActiveSeq := TO_STRING(THIS^.eSeq);

CASE THIS^.stSeqCtrlGeneral.eActiveSeqState OF
E_SEQ_GENERAL.READY:;

	
E_SEQ_GENERAL.EXECUTE:;
	IF TRUE
	THEN
		THIS^.stSeqCtrlGeneral.eActiveSeqState := E_SEQ_GENERAL.RESET;
	END_IF
  
E_SEQ_GENERAL.RESET:;
	THIS^.stSeqCtrlGeneral.iInternalSeqStateCase := 0;
	IF TRUE
	THEN
    THIS^.bResult := FALSE;
		THIS^.stSeqCtrlGeneral.eActiveSeqState := E_SEQ_GENERAL.BUSY;
	END_IF
  
E_SEQ_GENERAL.BUSY:;
	CASE THIS^.stSeqCtrlGeneral.iInternalSeqStateCase OF
		0:	// Entrance step --> Create command
      IF TRUE 
      AND THIS^.bAdsConnected
      AND NOT THIS^.bBusy
      AND THIS^.bReady
			THEN 
        THIS^.bWriteStructData := TRUE;
        THIS^.stSeqCtrlGeneral.iInternalSeqStateCase := 10;
			END_IF
      
    10:	// Wait for done
      IF TRUE 
      AND NOT THIS^.bBusy
      AND THIS^.bReady
      AND NOT THIS^.bWriteStructData
			THEN 
        THIS^.stSeqCtrlGeneral.iInternalSeqStateCase := 1000;
			END_IF
      
    1000: // Exit step
      IF TRUE
      THEN
        THIS^.stSeqCtrlGeneral.iInternalSeqStateCase := 9999;
			END_IF
      
	ELSE
		THIS^.stSeqCtrlGeneral.eActiveSeqState := E_SEQ_GENERAL.DONE;  
	END_CASE
	THIS^.stSeqCtrlGeneral.strExtraInfo := CONCAT('Internal state: ', TO_STRING(THIS^.stSeqCtrlGeneral.iInternalSeqStateCase));

E_SEQ_GENERAL.DONE:;

E_SEQ_GENERAL.ERROR:;

E_SEQ_GENERAL.TIME_OUT:; 
IF TRUE
AND THIS^.stSeqCtrlGeneral.bTimeOutActiveQuit 
THEN
  THIS^.stSeqCtrlGeneral.strExtraInfo := 'Bitte quittieren und erneut testen';
  IF TRUE
  //AND itfOpMode.P_QUIT
  THEN
    THIS^.stSeqCtrlGeneral.eActiveSeqState := E_SEQ_GENERAL.EXECUTE;
	END_IF
  
END_IF

ELSE
  THIS^.stSeqCtrlGeneral.eActiveSeqState := E_SEQ_GENERAL.ERROR;
END_CASE
END_METHOD

METHOD PRIVATE _m_SequenceManager
VAR_INPUT
END_VAR
IF FALSE
//AND THIS^.eActiveSeqState=DONE 
AND eLastSeq<>eSeq
THEN
	IF THIS^.stSeqCtrlGeneral.eActiveSeqState<>E_SEQ_GENERAL.EXECUTE THEN
		THIS^.stSeqCtrlGeneral.eActiveSeqState:=E_SEQ_GENERAL.READY;
	END_IF
END_IF

eSeq := eNextSeq;

//DelayTimer und TimeOut Timer verwalten
stSeqCtrlGeneral.bActiveStep:=	TRUE
				AND eLastSeq					=	eSeq
				AND stSeqCtrlGeneral.eLastActiveSeqState			=	stSeqCtrlGeneral.eActiveSeqState
				AND	stSeqCtrlGeneral.iLastInternalSeqStateCase	=	stSeqCtrlGeneral.iInternalSeqStateCase
				;
			
IF NOT stSeqCtrlGeneral.bActiveStep THEN
	stSeqCtrlGeneral.bDelayActive:=FALSE;
	stSeqCtrlGeneral.bTimeOutActiveQuit:=FALSE;
	stSeqCtrlGeneral.bTimeOutActiveNoQuit:=FALSE;
  THIS^.stSeqCtrlGeneral.strExtraInfo:='';
END_IF

_m_SaveLastStep();
stSeqCtrlGeneral.tonDelay	(IN:=stSeqCtrlGeneral.bActiveStep AND stSeqCtrlGeneral.bDelayActive, 		PT:=stSeqCtrlGeneral.tDelay);
stSeqCtrlGeneral.tonTimeOut	(IN:=stSeqCtrlGeneral.bActiveStep AND (stSeqCtrlGeneral.bTimeOutActiveNoQuit OR stSeqCtrlGeneral.bTimeOutActiveQuit), 	PT:=stSeqCtrlGeneral.tTimeOut);
stSeqCtrlGeneral.tonStepTime	(IN:= stSeqCtrlGeneral.bActiveStep, PT:= T#24H);

IF stSeqCtrlGeneral.tonTimeOut.Q  THEN
	stSeqCtrlGeneral.eActiveSeqState:=E_SEQ_GENERAL.TIME_OUT;
END_IF

IF stSeqCtrlGeneral.iError<>0 THEN
	eSeq:=E_SEQ_DATABASE.ERROR_SEQ;
END_IF



eLastSeq					:=	eSeq;
stSeqCtrlGeneral.eLastActiveSeqState			:=	stSeqCtrlGeneral.eActiveSeqState;
stSeqCtrlGeneral.iLastInternalSeqStateCase	:=	stSeqCtrlGeneral.iInternalSeqStateCase;

// Reset set ready state
IF THIS^.stSeqCtrlGeneral.bExitSetReadyState THEN
  THIS^.stSeqCtrlGeneral.bExitSetReadyState := FALSE;
END_IF
END_METHOD

METHOD PRIVATE _m_TimeOut : BOOL
VAR_INPUT
	bTimeoutActiveToQuit:	BOOL;
	bTimeOutActiveNoQuit:	BOOL;
	tTimeOut:				TIME;	
END_VAR
THIS^.stSeqCtrlGeneral.bTimeOutActiveQuit:=	bTimeoutActiveToQuit;
THIS^.stSeqCtrlGeneral.bTimeOutActiveNoQuit:=	bTimeOutActiveNoQuit;
THIS^.stSeqCtrlGeneral.tTimeOut:=			tTimeOut;
_m_TimeOut:=FALSE;
IF THIS^.stSeqCtrlGeneral.tonTimeOut.Q THEN
	_m_TimeOut:=TRUE;
END_IF
END_METHOD

ACTION A_010_ADSState:
tonADSState(IN:= NOT bResetADSStateTimer, PT:= tLifeBitTimeout);
bResetADSStateTimer := FALSE;
tonADSState.IN := TRUE;

CASE uiADSStateSeq OF
  0:
    IF bADSLifeBit AND bAdsConnected THEN
      bResetADSStateTimer := TRUE;
      bADSState := TRUE;
      uiADSStateSeq := 1;
    ELSIF tonADSState.Q THEN
      stSeqCtrlGeneral.eActiveSeqState := E_SEQ_GENERAL.ERROR;
      bADSState := FALSE;
		END_IF
  1:
    IF NOT bADSLifeBit AND bAdsConnected THEN
      bResetADSStateTimer := TRUE;
      bADSState := TRUE;
      uiADSStateSeq := 0;
    ELSIF tonADSState.Q THEN
      stSeqCtrlGeneral.eActiveSeqState := E_SEQ_GENERAL.ERROR;
      bADSState := FALSE;
		END_IF
END_CASE
END_ACTION

ACTION A_020_InfluxDBState:
tonInfluxDBState(IN:= NOT bResetInfluxDBStateTimer, PT:= tLifeBitTimeout);
bResetInfluxDBStateTimer := FALSE;
tonInfluxDBState.IN := TRUE;

CASE uiInfluxDBStateSeq OF
  0:
    IF bDBLifeBit AND bAdsConnected THEN
      bResetInfluxDBStateTimer := TRUE;
      bInfluxDBState := TRUE;
      uiInfluxDBStateSeq := 1;
    ELSIF tonInfluxDBState.Q THEN
      stSeqCtrlGeneral.eActiveSeqState := E_SEQ_GENERAL.ERROR;
      bInfluxDBState := FALSE;
		END_IF
  1:
    IF NOT bDBLifeBit AND bAdsConnected THEN
      bResetInfluxDBStateTimer := TRUE;
      bInfluxDBState := TRUE;
      uiInfluxDBStateSeq := 0;
    ELSIF tonInfluxDBState.Q THEN
      stSeqCtrlGeneral.eActiveSeqState := E_SEQ_GENERAL.ERROR;
      bInfluxDBState := FALSE;
		END_IF
END_CASE
END_ACTION

METHOD FB_init : BOOL
VAR_INPUT
	bInitRetains : BOOL; // if TRUE, the retain variables are initialized (warm start / cold start)
	bInCopyCode : BOOL;  // if TRUE, the instance afterwards gets moved into the copy code (online change)
  
  itfOpMode:											                        I_OP_MODE;  
  itfEventLogger:                                         I_EVENT_LOGGER;
END_VAR
THIS^.itfOpMode := itfOpMode;
THIS^.itfEventLogger := itfEventLogger;
END_METHOD

METHOD M_BucketExistCheck : BOOL
VAR_INPUT
	(* Name of the table that is to be read.*)
	sBucketName	: Tc2_System.T_MaxString;
END_VAR
VAR_OUTPUT
	(* Result*)
	bResult	: BOOL;
END_VAR
// Output
bResult := THIS^.bResult;

M_BucketExistCheck := THIS^.stSeqCtrlGeneral.eActiveSeqState = E_SEQ_GENERAL.DONE;

// Input
THIS^.sBucketName := sBucketName;

// General
IF THIS^.stSeqCtrlGeneral.eActiveSeqState = E_SEQ_GENERAL.READY THEN
  THIS^.eNextSeq := E_SEQ_DATABASE.BUCKET_EXIST_CHECK;
  THIS^.stSeqCtrlGeneral.eActiveSeqState := E_SEQ_GENERAL.EXECUTE;
END_IF
END_METHOD

METHOD M_ClearMeasurement : BOOL
VAR_INPUT
	(* Bucket name*)
	sBucketName	: Tc2_System.T_MaxString;
	(* Name of the measure to clear*)
	sMeasurementName	: Tc2_System.T_MaxString;
	(* From date time (Range)*)
	dtFrom	: DATE_AND_TIME;
	(* To date time (Range)*)
	dtTo	: DATE_AND_TIME;
END_VAR
VAR_OUTPUT
	(* Result*)
	bResult	: BOOL;
END_VAR
// Output
bResult := THIS^.bResult;

M_ClearMeasurement := THIS^.stSeqCtrlGeneral.eActiveSeqState = E_SEQ_GENERAL.DONE;

// Input
THIS^.sBucketName := sBucketName;
THIS^.sMeasurementName := sMeasurementName;
THIS^.dtFrom := dtFrom;
THIS^.dtTo := dtTo;

// General
IF THIS^.stSeqCtrlGeneral.eActiveSeqState = E_SEQ_GENERAL.READY THEN
  THIS^.eNextSeq := E_SEQ_DATABASE.CLEAR_MEASUREMENT;
  THIS^.stSeqCtrlGeneral.eActiveSeqState := E_SEQ_GENERAL.EXECUTE;
END_IF
END_METHOD

METHOD M_DeleteAllMeasurements : BOOL
VAR_INPUT
	(* Bucket name*)
	sBucketName	: Tc2_System.T_MaxString;
END_VAR
VAR_OUTPUT
	(* Result*)
	bResult	: BOOL;
END_VAR
// Output
bResult := THIS^.bResult;

M_DeleteAllMeasurements := THIS^.stSeqCtrlGeneral.eActiveSeqState = E_SEQ_GENERAL.DONE;

// Input
THIS^.sBucketName := sBucketName;

// General
IF THIS^.stSeqCtrlGeneral.eActiveSeqState = E_SEQ_GENERAL.READY THEN
  THIS^.eNextSeq := E_SEQ_DATABASE.DELETE_ALL_MEASUREMENTS;
  THIS^.stSeqCtrlGeneral.eActiveSeqState := E_SEQ_GENERAL.EXECUTE;
END_IF
END_METHOD

METHOD M_DeleteField : BOOL
VAR_INPUT
	(* Bucket name*)
	sBucketName	: Tc2_System.T_MaxString;
	(* Measurement Name*)
	sMeasurementName	: Tc2_System.T_MaxString;
	(* Tag Name*)
	sTagName	: Tc2_System.T_MaxString;
	(* Field Name*)
	sFieldName	: Tc2_System.T_MaxString;
END_VAR
VAR_OUTPUT
	(* Result*)
	bResult	: BOOL;
END_VAR
// Output
bResult := THIS^.bResult;

M_DeleteField := THIS^.stSeqCtrlGeneral.eActiveSeqState = E_SEQ_GENERAL.DONE;

// Input
THIS^.sBucketName := sBucketName;
THIS^.sMeasurementName := sMeasurementName;
THIS^.sTagName := sTagName;
THIS^.sFieldNameExistCheck := sFieldName;

// General
IF THIS^.stSeqCtrlGeneral.eActiveSeqState = E_SEQ_GENERAL.READY THEN
  THIS^.eNextSeq := E_SEQ_DATABASE.DELETE_FIELD;
  THIS^.stSeqCtrlGeneral.eActiveSeqState := E_SEQ_GENERAL.EXECUTE;
END_IF
END_METHOD

METHOD M_DeleteMeasurement : BOOL
VAR_INPUT
	(* Bucket name*)
	sBucketName	: Tc2_System.T_MaxString;
	(* Name of the measure to delete.*)
	sMeasurementName	: Tc2_System.T_MaxString;
END_VAR
VAR_OUTPUT
	(* Result*)
	bResult	: BOOL;
END_VAR
// Output
bResult := THIS^.bResult;

M_DeleteMeasurement := THIS^.stSeqCtrlGeneral.eActiveSeqState = E_SEQ_GENERAL.DONE;

// Input
THIS^.sBucketName := sBucketName;
THIS^.sMeasurementName := sMeasurementName;

// General
IF THIS^.stSeqCtrlGeneral.eActiveSeqState = E_SEQ_GENERAL.READY THEN
  THIS^.eNextSeq := E_SEQ_DATABASE.DELETE_MEASUREMENT;
  THIS^.stSeqCtrlGeneral.eActiveSeqState := E_SEQ_GENERAL.EXECUTE;
END_IF
END_METHOD

METHOD M_DeleteTag : BOOL
VAR_INPUT
	(* Bucket name*)
	sBucketName	: Tc2_System.T_MaxString;
	(* Measurement Name*)
	sMeasurementName	: Tc2_System.T_MaxString;
	(* Tag Name*)
	sTagName	: Tc2_System.T_MaxString;
END_VAR
VAR_OUTPUT
	(* Result*)
	bResult	: BOOL;
END_VAR
// Output
bResult := THIS^.bResult;

M_DeleteTag := THIS^.stSeqCtrlGeneral.eActiveSeqState = E_SEQ_GENERAL.DONE;

// Input
THIS^.sBucketName := sBucketName;
THIS^.sMeasurementName := sMeasurementName;
THIS^.sTagName := sTagName;

// General
IF THIS^.stSeqCtrlGeneral.eActiveSeqState = E_SEQ_GENERAL.READY THEN
  THIS^.eNextSeq := E_SEQ_DATABASE.DELETE_TAG;
  THIS^.stSeqCtrlGeneral.eActiveSeqState := E_SEQ_GENERAL.EXECUTE;
END_IF
END_METHOD

METHOD M_DeleteTagContentBlock : BOOL
VAR_INPUT
	(* Bucket name*)
	sBucketName	: Tc2_System.T_MaxString;
	(* Measurement Name*)
	sMeasurementName	: Tc2_System.T_MaxString;
	(* Tag Name*)
	sTagName	: Tc2_System.T_MaxString;
	(* Date and time from*)
	dtFrom	: DATE_AND_TIME;
	(* Date and Time to*)
	dtTo	: DATE_AND_TIME;
END_VAR
VAR_OUTPUT
	(* Result*)
	bResult	: BOOL;
END_VAR
// Output
bResult := THIS^.bResult;

M_DeleteTagContentBlock := THIS^.stSeqCtrlGeneral.eActiveSeqState = E_SEQ_GENERAL.DONE;

// Input
THIS^.sBucketName := sBucketName;
THIS^.sMeasurementName := sMeasurementName;
THIS^.sTagName := sTagName;
THIS^.dtFrom := dtFrom;
THIS^.dtTo := dtTo;

// General
IF THIS^.stSeqCtrlGeneral.eActiveSeqState = E_SEQ_GENERAL.READY THEN
  THIS^.eNextSeq := E_SEQ_DATABASE.DELETE_TAG_CONTENT_BLOCK;
  THIS^.stSeqCtrlGeneral.eActiveSeqState := E_SEQ_GENERAL.EXECUTE;
END_IF
END_METHOD

METHOD M_FieldExistCheck : BOOL
VAR_INPUT
	(* Bucket name*)
	sBucketName	: Tc2_System.T_MaxString;
	(* Measurement Name*)
	sMeasurementName	: Tc2_System.T_MaxString;
	(* Tag Name*)
	sTagName	: Tc2_System.T_MaxString;
	(* Field Name*)
	sFieldName	: Tc2_System.T_MaxString;
END_VAR
VAR_OUTPUT
	(* Result*)
	bResult	: BOOL;
END_VAR
// Output
bResult := THIS^.bResult;

M_FieldExistCheck := THIS^.stSeqCtrlGeneral.eActiveSeqState = E_SEQ_GENERAL.DONE;

// Input
THIS^.sBucketName := sBucketName;
THIS^.sMeasurementName := sMeasurementName;
THIS^.sTagName := sTagName;
THIS^.sFieldNameExistCheck := sFieldName;

// General
IF THIS^.stSeqCtrlGeneral.eActiveSeqState = E_SEQ_GENERAL.READY THEN
  THIS^.eNextSeq := E_SEQ_DATABASE.FIELD_EXIST_CHECK;
  THIS^.stSeqCtrlGeneral.eActiveSeqState := E_SEQ_GENERAL.EXECUTE;
END_IF
END_METHOD

METHOD M_GetTotalMeasurements : BOOL
VAR_INPUT
	(* Bucket name*)
	sBucketName	: Tc2_System.T_MaxString;
END_VAR
VAR_OUTPUT
  (* Process success*)
  bResult:    BOOL;
	(* Result value*)
	uiResult:   UINT;
END_VAR
// Output
bResult := THIS^.bResult;
uiResult := THIS^.uiTotalMeasurements;

M_GetTotalMeasurements := THIS^.stSeqCtrlGeneral.eActiveSeqState = E_SEQ_GENERAL.DONE;

// Input
THIS^.sBucketName := sBucketName;

// General
IF THIS^.stSeqCtrlGeneral.eActiveSeqState = E_SEQ_GENERAL.READY THEN
  THIS^.eNextSeq := E_SEQ_DATABASE.GET_TOTAL_MEASUREMENTS;
  THIS^.stSeqCtrlGeneral.eActiveSeqState := E_SEQ_GENERAL.EXECUTE;
END_IF
END_METHOD

METHOD M_MeasurementExistCheck : BOOL
VAR_INPUT
	(* Bucket name*)
	sBucketName	: Tc2_System.T_MaxString;
	(* Name of the table that is to be read.*)
	sMeasurementName	: Tc2_System.T_MaxString;
END_VAR
VAR_OUTPUT
	(* Result*)
	bResult	: BOOL;
END_VAR
// Output
bResult := THIS^.bResult;

M_MeasurementExistCheck := THIS^.stSeqCtrlGeneral.eActiveSeqState = E_SEQ_GENERAL.DONE;

// Input
THIS^.sBucketName := sBucketName;
THIS^.sMeasurementName := sMeasurementName;

// General
IF THIS^.stSeqCtrlGeneral.eActiveSeqState = E_SEQ_GENERAL.READY THEN
  THIS^.eNextSeq := E_SEQ_DATABASE.MEASUREMENT_EXIST_CHECK;
  THIS^.stSeqCtrlGeneral.eActiveSeqState := E_SEQ_GENERAL.EXECUTE;
END_IF
END_METHOD

METHOD M_Reset : BOOL
M_Reset := THIS^.stSeqCtrlGeneral.eActiveSeqState = E_SEQ_GENERAL.DONE;

// General
IF THIS^.stSeqCtrlGeneral.eActiveSeqState = E_SEQ_GENERAL.READY THEN
  THIS^.eNextSeq := E_SEQ_DATABASE.INIT;
  THIS^.stSeqCtrlGeneral.eActiveSeqState := E_SEQ_GENERAL.EXECUTE;
END_IF
END_METHOD

(*=== Method: M_Run  ============================================

 @brief: Here is the global code (Timer, Event, Flange,...)*)
METHOD M_Run
END_METHOD

METHOD M_SetReady : BOOL
VAR_INPUT
END_VAR
M_SetReady := TRUE
              AND THIS^.stSeqCtrlGeneral.eActiveSeqState = E_SEQ_GENERAL.READY
              AND THIS^.eSeq = E_SEQ_DATABASE.BASE;

THIS^.stSeqCtrlGeneral.eActiveSeqState := E_SEQ_GENERAL.READY;
THIS^.eNextSeq := E_SEQ_DATABASE.BASE;
END_METHOD

METHOD M_TagExistCheck : BOOL
VAR_INPUT
	(* Bucket name*)
	sBucketName	: Tc2_System.T_MaxString;
	(* Measurement Name*)
	sMeasurementName	: Tc2_System.T_MaxString;
	(* Tag Name*)
	sTagName	: Tc2_System.T_MaxString;
END_VAR
VAR_OUTPUT
	(* Result*)
	bResult	: BOOL;
END_VAR
// Output
bResult := THIS^.bResult;

M_TagExistCheck := THIS^.stSeqCtrlGeneral.eActiveSeqState = E_SEQ_GENERAL.DONE;

// Input
THIS^.sBucketName := sBucketName;
THIS^.sMeasurementName := sMeasurementName;
THIS^.sTagName := sTagName;

// General
IF THIS^.stSeqCtrlGeneral.eActiveSeqState = E_SEQ_GENERAL.READY THEN
  THIS^.eNextSeq := E_SEQ_DATABASE.TAG_EXIST_CHECK;
  THIS^.stSeqCtrlGeneral.eActiveSeqState := E_SEQ_GENERAL.EXECUTE;
END_IF
END_METHOD

METHOD M_WriteStruct : BOOL
VAR_INPUT
	(* Bucket name*)
	sBucketName:                  T_MaxString;
	(* Name of the table that is to be read.*)
	sMeasurementName:             T_MaxString;
	(* Tag name*)
	sTagName:                     T_MaxString;
  (* Field values list*)
	stFieldValues:                ST_DATABASE_RECORD;
  (* Field struct content (Variable names) *)
  //pFieldStructContent:          POINTER TO ARRAY [0..99] OF T_MaxString;
	(* Field names list: names that appear in the database*)
	//pFieldNames:                  POINTER TO ARRAY [0..99] OF T_MaxString;
END_VAR
VAR_OUTPUT
	(* Result*)
	bResult	: BOOL;
END_VAR
// Output
bResult := THIS^.bResult;

M_WriteStruct := THIS^.stSeqCtrlGeneral.eActiveSeqState = E_SEQ_GENERAL.DONE;

// Input
THIS^.sBucketName := sBucketName;
THIS^.sMeasurementName := sMeasurementName;
THIS^.sTagName := sTagName;
THIS^.stFieldValues := stFieldValues;
//THIS^.pFieldStructContent := pFieldStructContent;
//THIS^.pFieldNames := pFieldNames;



// General
IF THIS^.stSeqCtrlGeneral.eActiveSeqState = E_SEQ_GENERAL.READY THEN
  THIS^.eNextSeq := E_SEQ_DATABASE.WRITE_STRUCT;
  THIS^.stSeqCtrlGeneral.eActiveSeqState := E_SEQ_GENERAL.EXECUTE;
END_IF
END_METHOD

PROPERTY P_ADSLifebit : BOOL
GET
P_ADSLifebit := THIS^.bADSLifeBit;
END_GET
END_PROPERTY

{warning 'Eigenschaftenimplementierung hinzufügen'}
PROPERTY P_ADSState : BOOL
GET
P_ADSState := THIS^.bADSState;
END_GET
END_PROPERTY

PROPERTY P_Connected : BOOL
GET
P_Connected := false;
END_GET
END_PROPERTY

{warning 'Eigenschaftenimplementierung hinzufügen'}
PROPERTY P_Error : BOOL
GET
P_Error := THIS^.stSeqCtrlGeneral.eActiveSeqState = E_SEQ_GENERAL.ERROR;
END_GET
END_PROPERTY

{warning 'Eigenschaftenimplementierung hinzufügen'}
(*=== Property: P_Event  ============================================

 @param [set]: 	Set the Structure "ST_EVENT" from another Object
 @param [get]: 	Return the Structure "ST_EVENT", it contains the actual 
					event of the Object *)
PROPERTY P_Event : GenLib.ST_EVENT
GET
END_GET
SET
END_SET
END_PROPERTY

{warning 'Eigenschaftenimplementierung hinzufügen'}
(*=== Property: P_FullObjectPath  ============================================

 @param [set]: 	Set the Object Path (Clear String of Object)
 @param [get]: 	Return the Objectpath *)
PROPERTY P_FullObjectPath : STRING
GET
P_FullObjectPath:= THIS^.strFullObjectPath;
END_GET
SET
THIS^.strFullObjectPath:=P_FullObjectPath;
END_SET
END_PROPERTY

{warning 'Eigenschaftenimplementierung hinzufügen'}
(*=== Property: P_Global_Ack  ============================================

 @param [set]: 	Set the Bit for Ack from another Object
 @param [get]: 	Return the state of Ack Bit*)
PROPERTY P_Global_Ack : BOOL
GET
END_GET
SET
END_SET
END_PROPERTY

{warning 'Eigenschaftenimplementierung hinzufügen'}
(*=== Property: P_GlobalID  ============================================

 @param [set]: 	-
 @param [get]: 	Return the string of instance path*)
PROPERTY P_GlobalID : STRING
GET
P_GlobalID:= THIS^.strInstancePath;
END_GET
END_PROPERTY

{warning 'Eigenschaftenimplementierung hinzufügen'}
PROPERTY P_InfluxDBLifeBit : BOOL
GET
P_InfluxDBLifeBit := THIS^.bDBLifeBit;
END_GET
END_PROPERTY

PROPERTY P_InfluxDBState : BOOL
GET
P_InfluxDBState := THIS^.bInfluxDBState;
END_GET
END_PROPERTY

END_FUNCTION_BLOCK

(* stored: Version 1.1.0.1, ProductVersion 3.1.4024.12
   POU FB_INFLUX_DB_ADS: Id {737bb810-17d3-41b2-ad6b-a6b9cc0fb535}, SpecialFunc None
   Folder ACTIONS: Id {0a706a70-b10d-4937-b0fe-eb1d297f5b0d}
   Folder PRIVAT: Id {04526e9c-1367-468a-9725-50f7bcef8cff}
   Folder SEQUENCE: Id {5a90cded-5971-42c2-9668-0b858782d80f}
   Method _m_DebugManager: Id {f060f21f-c204-4398-89fd-4c195c9da6a2}
   Method _m_Delay: Id {fb17f725-cb65-4789-8c5a-5a0a1fa45055}
   Method _m_GeneralStepSetting: Id {4ae7e319-36c6-45ef-90c1-5f8bdda48041}
   Method _m_SaveLastStep: Id {eb38dcf2-f9cd-4646-8def-1027668199c7}
   Method _m_Seq_BUCKET_EXIST_CHECK: Id {4e475998-cbfd-430a-856a-fdb3281ac526}
   Method _m_Seq_CLEAR_MEASUREMENT: Id {b92cf6ef-876b-49e9-bde6-775be015f5af}
   Method _m_Seq_DELETE_ALL_MEASUREMENTS: Id {9868a3f2-9899-4ba5-8b91-09d47c1fec7e}
   Method _m_Seq_DELETE_FIELD: Id {226fd484-7c1a-4bb0-8131-f214c1586370}
   Method _m_Seq_DELETE_MEASUREMENT: Id {e0b18201-b710-43fc-8564-6a27e4c0747b}
   Method _m_Seq_DELETE_TAG: Id {0d551c7e-a4bb-4575-b494-3b749ab42118}
   Method _m_Seq_DELETE_TAG_CONTENT_BLOCK: Id {e12ba077-6828-4185-b3b9-654377707dcb}
   Method _m_Seq_FIELD_EXIST_CHECK: Id {2c2c8c0a-30f8-4ef7-a0bd-8564c914a89d}
   Method _m_Seq_GET_TOTAL_MEASUREMENTS: Id {558cc239-6d34-43a1-a4c9-b6e51e8ee745}
   Method _m_Seq_INIT: Id {1a4092c0-069d-44a5-9015-ede7594fe692}
   Method _m_Seq_MEASUREMENT_EXIST_CHECK: Id {ee65c0c1-175c-4046-a8fb-e4ae7eb1120b}
   Method _m_Seq_TAG_EXIST_CHECK: Id {bd2960d4-1656-40ee-a3df-dd762425b886}
   Method _m_Seq_WRITE_STRUCT: Id {f470c48c-229c-48c8-b99b-8a20c064ba52}
   Method _m_SequenceManager: Id {f06585bc-454f-440c-a615-f294a1de9843}
   Method _m_TimeOut: Id {6aca30a3-ccc2-46d4-951f-6b9d8fd454f9}
   Action A_010_ADSState: Id {e7a72e72-c00d-4af3-af01-148357e07b31}
   Action A_020_InfluxDBState: Id {af1680db-4575-4733-b039-2d5ef224709c}
   Method FB_init: Id {aeb12498-62e3-4e82-a75b-5428c8304956}
   Method M_BucketExistCheck: Id {263a11c2-ac1d-4257-a335-5278c769983c}
   Method M_ClearMeasurement: Id {8228e032-68a4-4513-8c36-fdc91174af11}
   Method M_DeleteAllMeasurements: Id {d1caf4f7-5e50-4d34-8cc3-b2287255f86d}
   Method M_DeleteField: Id {718bec70-73e6-4142-b061-f1f2292b6d6c}
   Method M_DeleteMeasurement: Id {a48ed3a1-2962-44da-8ccd-93cc8d663b07}
   Method M_DeleteTag: Id {ac9ac39d-706b-48d8-bb99-aaf8c40192ea}
   Method M_DeleteTagContentBlock: Id {d3ab90cf-47d4-4041-8f2a-6640dd63d064}
   Method M_FieldExistCheck: Id {61ded7b2-bc3b-45d4-b751-239631cc30e8}
   Method M_GetTotalMeasurements: Id {d0c66e1f-36a0-4f3e-be9f-5098c66bf484}
   Method M_MeasurementExistCheck: Id {fe04a21d-bbe3-4e97-a2f1-a5ffdb114224}
   Method M_Reset: Id {6a213e47-6369-4f7b-b2fa-5c224c780f2c}
   Method M_Run: Id {1f2b263a-9e93-4bf6-847b-1d760edaedae}
   Method M_SetReady: Id {b722e4e8-f5ee-43b9-888d-7efba6cba399}
   Method M_TagExistCheck: Id {a8a6bfdd-08ab-406d-ab58-01415266b01b}
   Method M_WriteStruct: Id {13475132-cd21-4d84-a07b-671cc309bb75}
   Property P_ADSLifebit: Id {b659c962-931e-47ff-a70f-529e182d0645}
   Get Get: Id {70be6309-f587-445e-8319-d8ae2eaf3196}
   Property P_ADSState: Id {52105ba9-74c0-47c0-b1ac-959c2db118d1}
   Get Get: Id {81a92754-6f97-4607-a2fb-fc8d9426c5ee}
   Property P_Connected: Id {e2a34010-e364-4b55-b704-962cbf3f9556}
   Get Get: Id {c91dfbfb-fb05-48d4-ab70-06073ef043f1}
   Property P_Error: Id {7213f8e5-eb43-44b7-896d-a75911420df4}
   Get Get: Id {391d443c-624a-4ad9-a747-2168458efc85}
   Property P_Event: Id {599a7f30-377c-4160-9921-65502e4028a7}
   Get Get: Id {339a6a8d-cb15-4679-a50d-3bde1faf7afa}
   Set Set: Id {6e14c6d9-48cb-4f90-a4fe-de51ba05bc69}
   Property P_FullObjectPath: Id {4bce0f63-8592-4d9a-9cea-3c9a77ec1fd4}
   Get Get: Id {7609d32b-79b2-4714-adf7-f62bf9c4ac7d}
   Set Set: Id {10de4671-7ae8-429c-82ff-7e5ae3ce9c72}
   Property P_Global_Ack: Id {51f9b3cd-90ba-4d57-bc68-fcc641f328ac}
   Get Get: Id {ebeec235-a651-4ff8-9090-403c5e7b7a33}
   Set Set: Id {78768363-d530-4a9f-a494-cc3888a36754}
   Property P_GlobalID: Id {5d6734d4-07cc-40b8-9f91-16b18999f2e6}
   Get Get: Id {58ddb13c-6848-4224-87aa-f535c7f33dce}
   Property P_InfluxDBLifeBit: Id {c8e364f7-26c0-445c-959d-95b6cb55f542}
   Get Get: Id {5e4c036e-c94d-49d8-88ba-f4534eb77348}
   Property P_InfluxDBState: Id {b602fa03-375a-4965-ac1e-cceeedec19ca}
   Get Get: Id {6fedc0c9-888d-413c-819b-80fcfd7e68fc} *)
